GLOBALCONSTANTS ADDRESS (* Global constants *)
  (* Standard: 61499-1 *)
  (* Version 1.0, 2025-09-04, Franz Höpfinger *)
  PACKAGE isobus::pgn;
  VAR_GLOBAL CONSTANT
    NULL_A : BYTE := 254; (* SAs with special meaning *)
    GLOBAL_A : INT := 255; (* < \brief 0xFEu NULL address - only sender with network man. *)
  END_VAR
END_GLOBALCONSTANTS
